TYPE ST_XV03_PerformanceDiagnosis :
STRUCT
	UL_UV_UNDERRNAGE_OR_UL_OV_OVERRANGE : BOOL;
	UA_OVERRANGE						: BOOL;
	OPEN_LOAD_AT_VALVE_COIL				: BOOL;
	SHORT_CIRCUIT_AT_VALVE_COIL			: BOOL;
	HWE									: BOOL;
END_STRUCT
END_TYPE

(* stored: Version 1.1.0.1, ProductVersion 3.1.4024.13
   DUT ST_XV03_PerformanceDiagnosis: Id {766f2e86-b41d-0996-14cf-914f2aa113b4} *)
